// Mitsubishi GX Works2 project: project part 2   PLC: FX3G

// global labels: Global1
VAR_GLOBAL
  switch1 AT X007 : BOOL;
  counter_start_day_result AT CS0 : BOOL;
  creamValue : REAL;  (* ערך למיכל קצפת *)
  creamTank AT D1100 : REAL;  (* ערך למיכל קצפת *)
  chocolateValue : REAL;  (* מיכל שוקולד *)
  chocolateTank AT D1102 : REAL;  (* מיכל השוקולד *)
  biscuitValue : REAL;  (* מיכל ביסקוויטים *)
  biscuitTank AT D1104 : REAL;  (* מיכל ביסקוויטים *)
  zilufTank AT D1112 : REAL;  (* ערך למיכל זילוף *)
END_VAR
VAR_GLOBAL CONSTANT
  zilufValue : REAL;  (* ערך למיכל זילוף *)
  dippingValue : REAL;  (* ערך למיכל טבילה *)
END_VAR
VAR_GLOBAL
  dippingTank AT D1114 : REAL;  (* ערך למיכל טבילה *)
END_VAR
VAR_GLOBAL CONSTANT
  unitsAmount : REAL;  (* כמות קרמבו מוכנים *)
END_VAR
VAR_GLOBAL
  amountDone AT D1118 : REAL;  (* כמות קרמבו מוכנים *)
  switch3 AT X011 : BOOL;  (* העברת הקצפת למיכל זילוף *)
END_VAR
VAR_GLOBAL CONSTANT
  creamInv : REAL := 700;  (* מלאי קצפת *)
END_VAR
VAR_GLOBAL
  courrentCream AT D1106 : REAL;
  curentCream AT D1106 : REAL;
  curentChoclate AT D1108 : REAL;
  curentBiscu AT D1110 : REAL;
END_VAR
VAR_GLOBAL CONSTANT
  chocolateInv : REAL := 500.0;  (* מלאי שוקולד *)
  constBisc : REAL := 6;
  contCream : REAL := 300;
END_VAR
VAR_GLOBAL
  switch4 AT X010 : BOOL;
  switch6 AT X005 : BOOL;
  ReadyToZiluf AT M0 : BOOL;
  TempBelow15 AT M1 : BOOL;
  ingReady AT Y000 : BOOL;
  sen_surface AT X003 : BOOL;
  switch7 AT X001 : BOOL;
  switch8 AT X002 : BOOL;
  under15 AT X001 : BOOL;
  under30 AT X002 : BOOL;
  zilufLight AT Y004 : BOOL;
  sen_camera AT X004 : BOOL;
  checkInv AT X011 : BOOL;  (* האם יש מספיק קצפת וביסקוויטים עבור זילוף *)
  enoughCream AT M111 : BOOL;
  notEnoughCream AT M150 : BOOL;
  enoughBisc AT M112 : BOOL;
  notEnoughBisc AT M151 : BOOL;
  dayStarted AT Y007 : BOOL;
  startDaySwitch AT X007 : BOOL;
  updateInventory AT CS0 : BOOL;
  enoughIng AT M113 : BOOL;
  startFlickering AT M0 : BOOL;
  Timer3 AT TC2 : BOOL;
  Timer1 AT TC1 : BOOL;
END_VAR
VAR_GLOBAL CONSTANT
  fourSeconds : INT := 5;
END_VAR
VAR_GLOBAL
  Timer2 AT TS1 : BOOL;
  Timer4 AT TS2 : BOOL;
  switch10 AT Y000 : BOOL;
  switch11 AT Y001 : BOOL;
  goToMachineB AT M130 : BOOL;
  Timer0 AT TC0 : BOOL;
END_VAR
VAR_GLOBAL CONSTANT
  countFour : INT := 40;
  countHalfSec : INT := 5;
END_VAR
VAR_GLOBAL
  Timer0_0 AT TS0 : BOOL;
  finishedZiluf AT M114 : BOOL;
  finished_fourSec_timer AT TS0 : BOOL;
  startZilufMachine AT X011 : BOOL;
  enoughIng_StartDay AT M115 : BOOL;
  Try_startDay AT M7 : BOOL;
  sample_analogIinput1 AT X006 : BOOL;
  sample AT X006 : BOOL;
END_VAR
VAR_GLOBAL CONSTANT
  normalize_val : INT := 390;
END_VAR
VAR_GLOBAL
  save_analog_val AT D8000 : INT;
  analog_input_chocolate AT D8280 : INT;
  coating AT M116 : BOOL;
  choose_coating_indicator AT M116 : BOOL;
END_VAR
VAR_GLOBAL CONSTANT
  bottom_limit_reg_coat : INT;  (* בדיקה האם הערך גדול מ0 *)
  upper_limit_reg_coat : INT := 5;
END_VAR
VAR_GLOBAL
  biggerThen_0 AT M118 : BOOL;
  smallerThen_5 AT M119 : BOOL;
END_VAR
VAR_GLOBAL CONSTANT
  bottom_limit_double_coat : INT := 6;  (* בדיקה האם הערך גדול 6 *)
END_VAR
VAR_GLOBAL
  biggerThen_6 AT M120 : BOOL;
END_VAR
VAR_GLOBAL CONSTANT
  upper_limit_double_coat : INT := 10;
END_VAR
VAR_GLOBAL
  smallerThen_10 AT M121 : BOOL;
  Regular_coat AT M122 : BOOL;
  Double_coat AT M123 : BOOL;
  successTranfer_toZiluf AT M125 : BOOL;
  chocolateInput AT D1117 : INT;
END_VAR
VAR_GLOBAL CONSTANT
  regularQuantity : REAL := 120;
  doubleQuantity : REAL := 240;
END_VAR
VAR_GLOBAL
  finished_transfer_toDipping AT M124 : BOOL;
  dippingIsOn AT Y003 : BOOL;
  TimerForDipping AT TC3 : BOOL;
END_VAR
VAR_GLOBAL CONSTANT
  countForDipping : INT := 50;
END_VAR
VAR_GLOBAL
  finishedDipping_timer AT TS3 : BOOL;
  enoughChocolate AT M126 : BOOL;  (* מספיק שוקולד לציפוי כפול *)
  notEnoughChocolate AT M128 : BOOL;
  stopDay AT M129 : BOOL;
END_VAR
VAR_GLOBAL CONSTANT
  initVakue : INT;
  initValue : REAL;
END_VAR
VAR_GLOBAL
  Timer_stopDay AT TC5 : BOOL;
END_VAR
VAR_GLOBAL CONSTANT
  countThreeSec : INT := 30;
END_VAR
VAR_GLOBAL
  finished_threeSec_timer AT TS5 : BOOL;
  TimerHalfSec AT TC4 : BOOL;
  finishHalfSec AT TS4 : BOOL;  (* סיום ציפוי *)
  countAgain AT M131 : BOOL;
  TimerHalfSec2 AT TC6 : BOOL;
  finishHalfSec2 AT TS6 : BOOL;
  fictiveLight AT M132 : BOOL;
  check2222 AT Y005 : BOOL;
  check1111 AT Y006 : BOOL;
  turnOnMachinA AT M142 : BOOL;
  stopDay_ind AT M140 : BOOL;
  packOne AT X000 : BOOL;  (* אריזת קרמבו בודד *)
  countPack AT CC1 : BOOL;
END_VAR
VAR_GLOBAL CONSTANT
  count_five : INT := 5;
END_VAR
VAR_GLOBAL
  countPack2 AT CC2 : BOOL;
END_VAR
VAR_GLOBAL CONSTANT
  count_six : INT := 6;
END_VAR
VAR_GLOBAL
  finish_pack5 AT CS1 : BOOL;
  almost_finishPack AT Y002 : BOOL;
  finish_pack6 AT CS2 : BOOL;
  countFinished_units AT CC3 : BOOL;
END_VAR
VAR_GLOBAL CONSTANT
  CountOne : INT := 1;
  add_one : REAL := 1;
END_VAR
VAR_GLOBAL
  Reset_C1 AT CC1 : BOOL;
  Reset_C2 AT CC2 : BOOL;
END_VAR
VAR_GLOBAL CONSTANT
  div_ten : REAL := 10;
  MUL_390 : REAL := 390;
END_VAR
VAR_GLOBAL
  finishDip AT M141 : BOOL;
  analog_output_save AT D8001 : REAL;
  savedAmount AT M133 : BOOL;
  amountDone_div AT D1119 : REAL;  (* כמות קרמבו מוכנים *)
  output_analog AT D8282 : INT;
  amountDone_int AT D1121 : INT;
  readyToStartMachineB AT M144 : BOOL;
  finished_dipping AT M145 : BOOL;
END_VAR

// task Task_01 (event TRUE, interval 0, priority 31): POU_01

PROGRAM POU_01
VAR CONSTANT
  biscInv : REAL := 100;  (* מלאי ביסקוויטים *)
END_VAR
VAR
  analog_input1 : INT;
END_VAR
VAR CONSTANT
  normal_chocolate : INT := 390;
END_VAR
(* structured ladder/FBD written out as ST: instructions are called as NAME(EN, inputs, outputs); _pN, _eN, _tN stand for wires *)
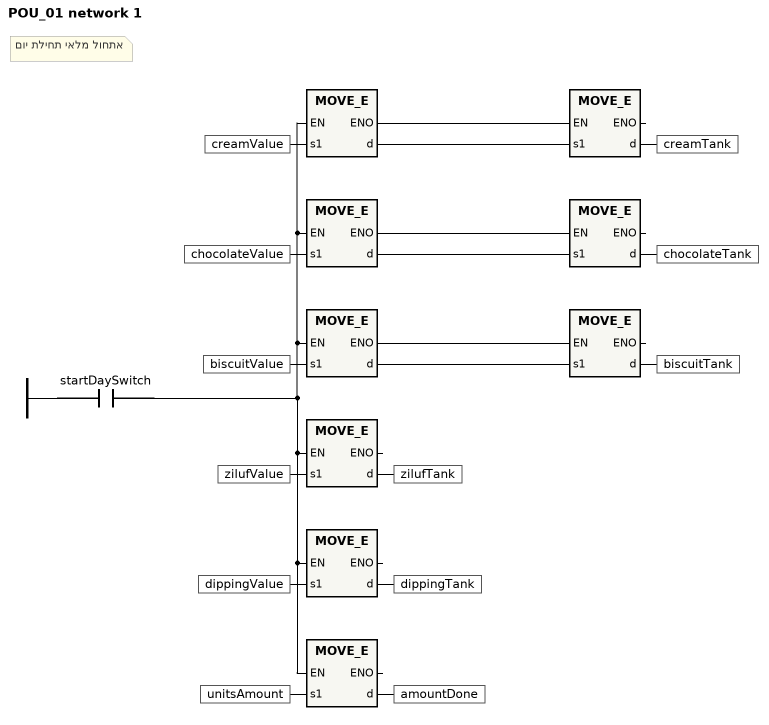
(* network 1 *)
(* אתחול מלאי תחילת יום *)
_e2 := MOVE_E(startDaySwitch, creamValue, _t1);
MOVE_E(_e2, _t1, creamTank);
_e4 := MOVE_E(startDaySwitch, chocolateValue, _t3);
MOVE_E(_e4, _t3, chocolateTank);
_e6 := MOVE_E(startDaySwitch, biscuitValue, _t5);
MOVE_E(_e6, _t5, biscuitTank);
MOVE_E(startDaySwitch, zilufValue, zilufTank);
MOVE_E(startDaySwitch, dippingValue, dippingTank);
MOVE_E(startDaySwitch, unitsAmount, amountDone);
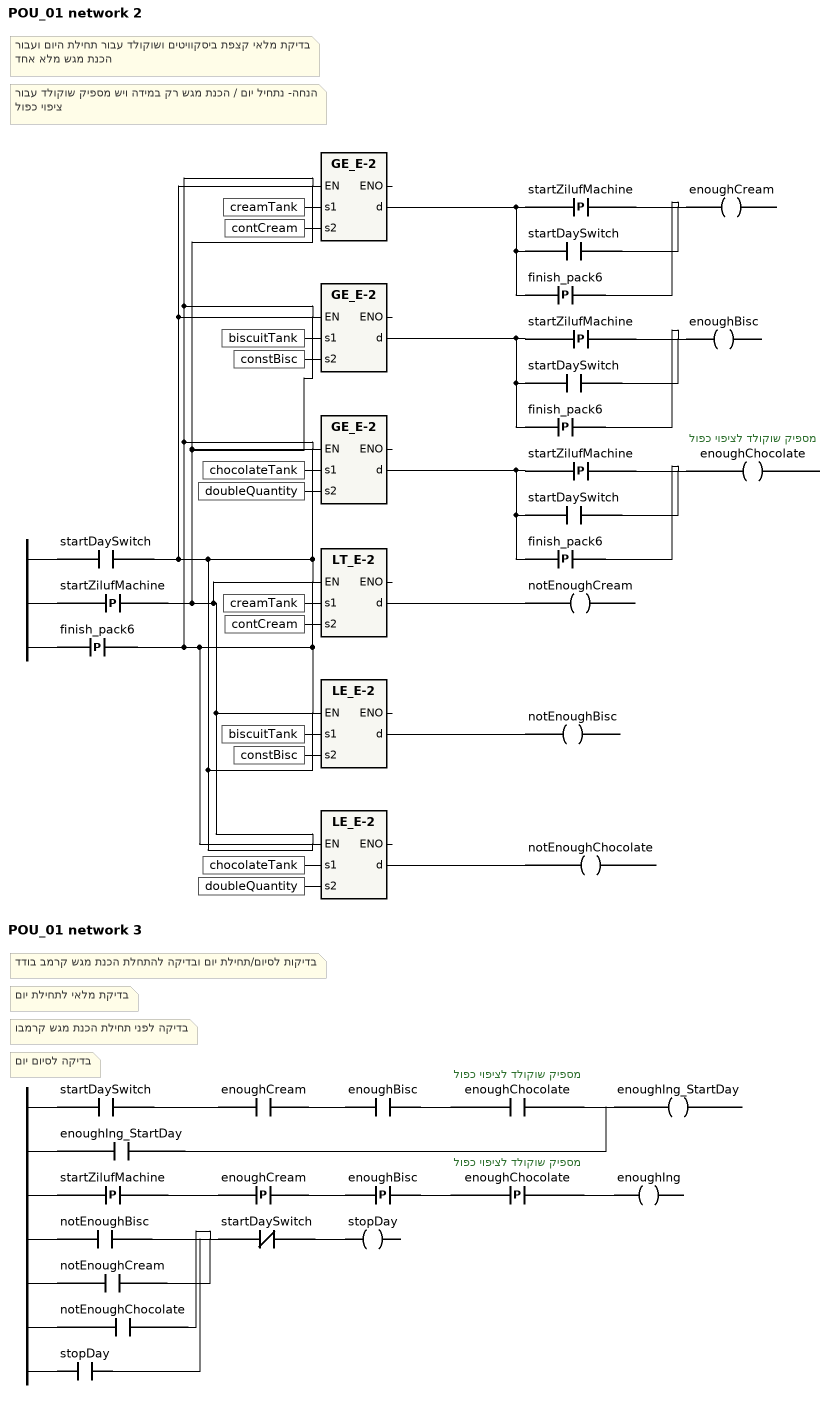
(* network 2 *)
(* בדיקת מלאי קצפת ביסקוויטים ושוקולד עבור תחילת היום ועבור הכנת מגש מלא אחד *)
(* הנחה- נתחיל יום / הכנת מגש רק במידה ויש מספיק שוקולד עבור ציפוי כפול *)
_p1 := startDaySwitch OR LDP(TRUE, startZilufMachine) OR LDP(TRUE, finish_pack6);
GE_E(_p1, creamTank, contCream, _t2);
enoughCream := (_t2 AND LDP(TRUE, startZilufMachine)) OR (_t2 AND startDaySwitch) OR (_t2 AND LDP(TRUE, finish_pack6));
LT_E(_p1, creamTank, contCream, _t3);
notEnoughCream := _t3;
GE_E(_p1, biscuitTank, constBisc, _t4);
enoughBisc := (_t4 AND LDP(TRUE, startZilufMachine)) OR (_t4 AND startDaySwitch) OR (_t4 AND LDP(TRUE, finish_pack6));
LE_E(_p1, biscuitTank, constBisc, _t5);
notEnoughBisc := _t5;
LE_E(_p1, chocolateTank, doubleQuantity, _t6);
notEnoughChocolate := _t6;
GE_E(_p1, chocolateTank, doubleQuantity, _t7);
enoughChocolate := (_t7 AND LDP(TRUE, startZilufMachine)) OR (_t7 AND startDaySwitch) OR (_t7 AND LDP(TRUE, finish_pack6));
(* network 3 *)
(* בדיקות לסיום/תחילת יום ובדיקה להתחלת הכנת מגש קרמב בודד *)
(* בדיקת מלאי לתחילת יום *)
(* בדיקה לפני תחילת הכנת מגש קרמבו *)
(* בדיקה לסיום יום *)
enoughIng_StartDay := (startDaySwitch AND enoughCream AND enoughBisc AND enoughChocolate) OR enoughIng_StartDay;
enoughIng := LDP(TRUE, startZilufMachine) AND LDP(TRUE, enoughCream) AND LDP(TRUE, enoughBisc) AND LDP(TRUE, enoughChocolate);
stopDay := (notEnoughBisc OR notEnoughCream OR notEnoughChocolate OR stopDay) AND NOT startDaySwitch;
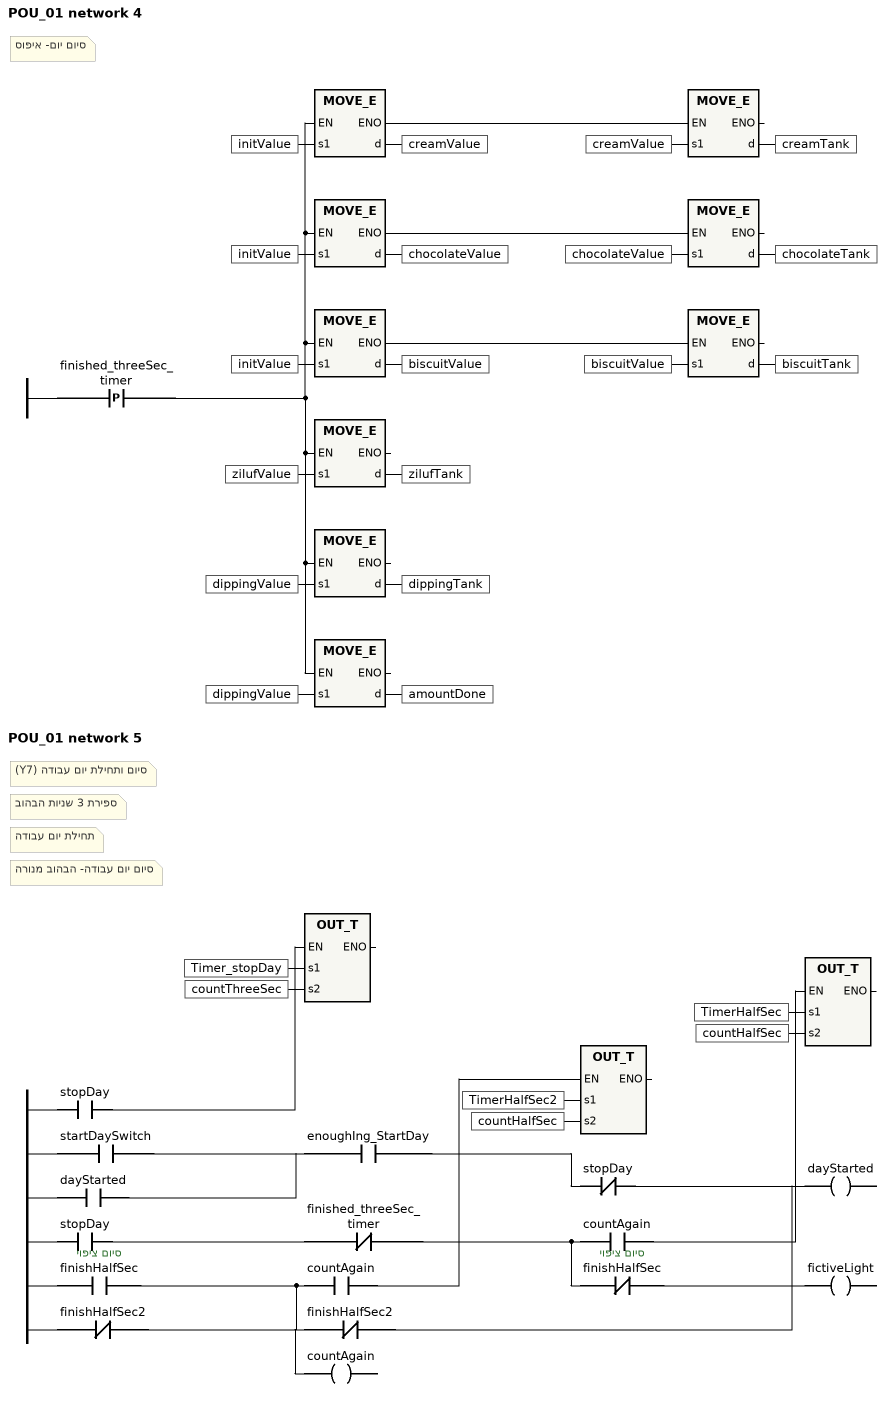
(* network 4 *)
(* סיום יום- איפוס *)
_p1 := LDP(TRUE, finished_threeSec_timer);
_e2 := MOVE_E(_p1, initValue, creamValue);
MOVE_E(_e2, creamValue, creamTank);
_e3 := MOVE_E(_p1, initValue, chocolateValue);
MOVE_E(_e3, chocolateValue, chocolateTank);
_e4 := MOVE_E(_p1, initValue, biscuitValue);
MOVE_E(_e4, biscuitValue, biscuitTank);
MOVE_E(_p1, zilufValue, zilufTank);
MOVE_E(_p1, dippingValue, dippingTank);
MOVE_E(_p1, dippingValue, amountDone);
(* network 5 *)
(* סיום ותחילת יום עבודה (Y7) *)
(* ספירת 3 שניות הבהוב *)
(* תחילת יום עבודה *)
(* סיום יום עבודה- הבהוב מנורה *)
OUT_T(stopDay, Timer_stopDay, countThreeSec);
dayStarted := (((startDaySwitch OR dayStarted) AND enoughIng_StartDay) AND NOT stopDay) OR (finishHalfSec AND NOT finishHalfSec2);
_p1 := stopDay AND NOT finished_threeSec_timer;
OUT_T(_p1 AND countAgain, TimerHalfSec, countHalfSec);
fictiveLight := _p1 AND NOT finishHalfSec;
OUT_T(finishHalfSec AND countAgain, TimerHalfSec2, countHalfSec);
countAgain := NOT finishHalfSec2;
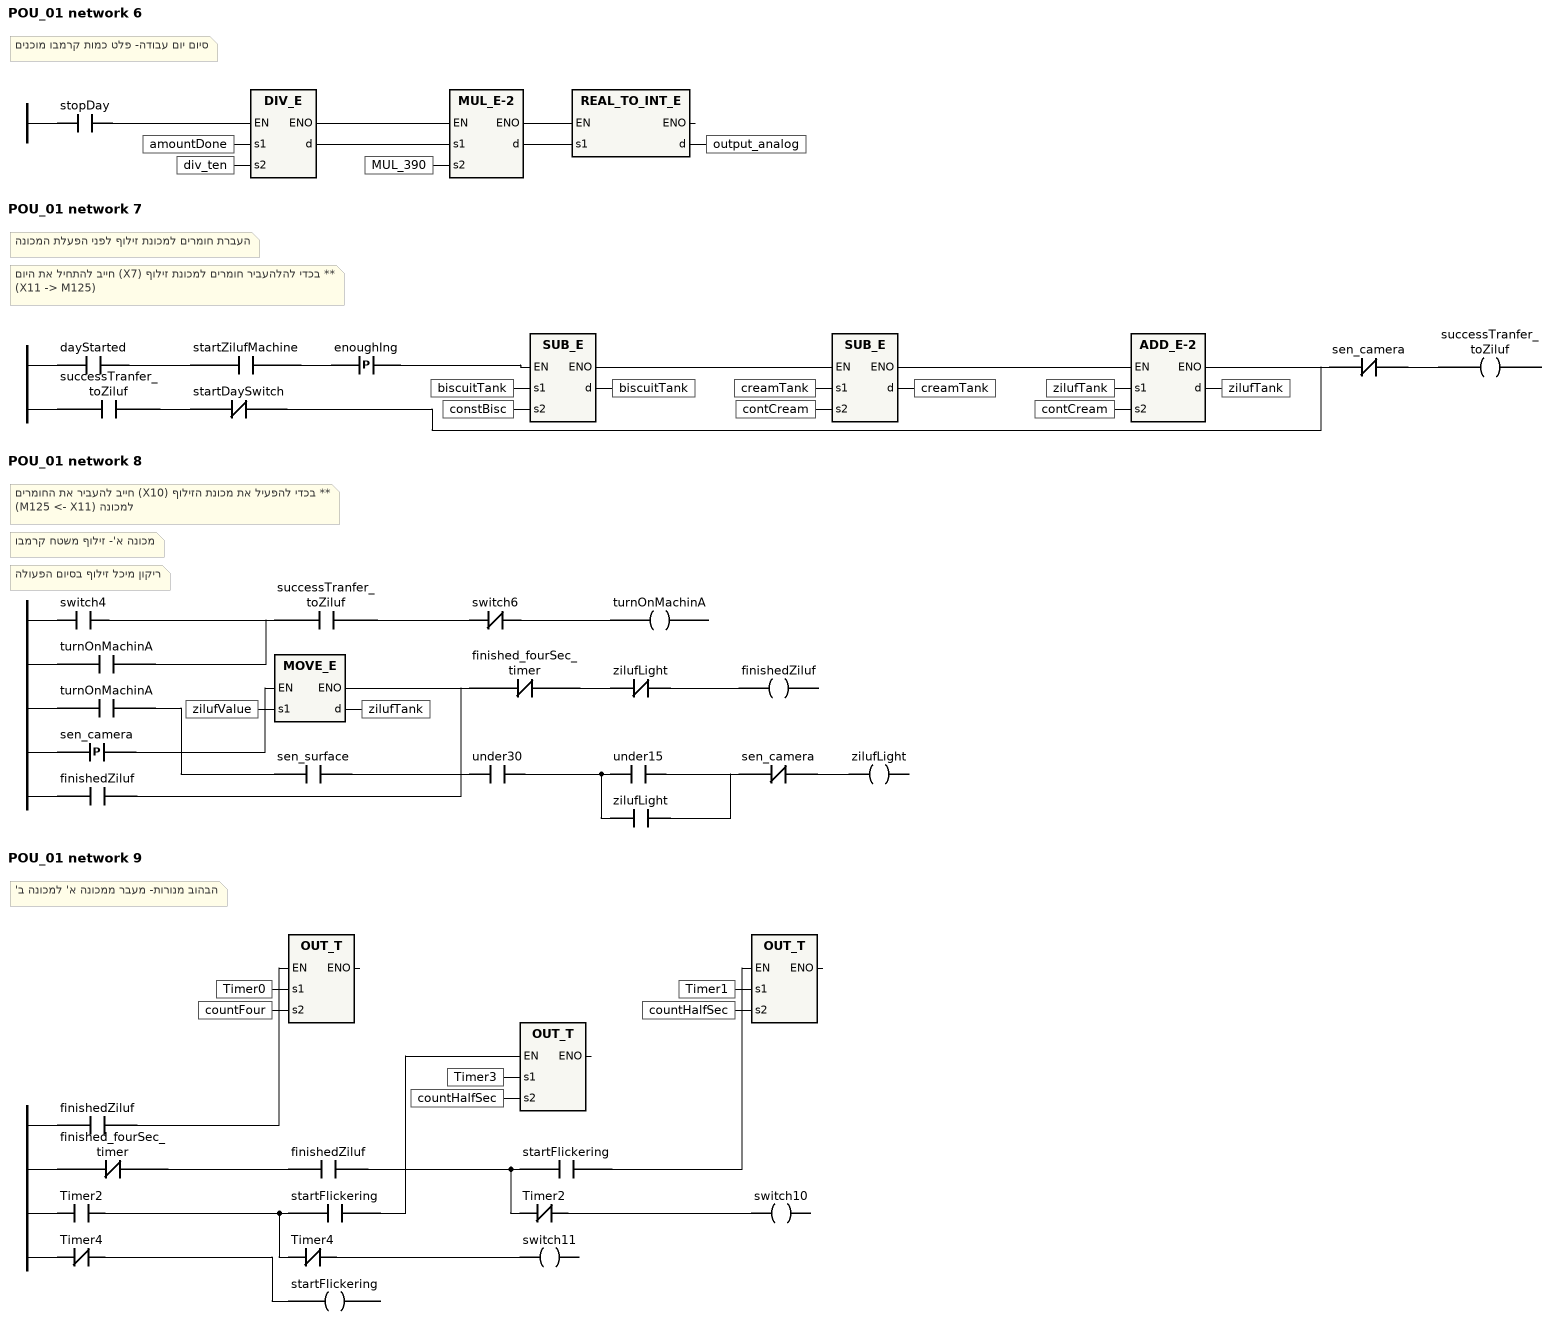
(* network 6 *)
(* סיום יום עבודה- פלט כמות קרמבו מוכנים *)
_e2 := DIV_E(stopDay, amountDone, div_ten, _t1);
_e4 := MUL_E(_e2, _t1, MUL_390, _t3);
REAL_TO_INT_E(_e4, _t3, output_analog);
(* network 7 *)
(* העברת חומרים למכונת זילוף לפני הפעלת המכונה *)
(* ** בכדי להלהעביר חומרים למכונת זילוף (X7) חייב להתחיל את היום  (X11 -> M125) *)
_e1 := SUB_E(dayStarted AND startZilufMachine AND LDP(TRUE, enoughIng), biscuitTank, constBisc, biscuitTank);
_e2 := SUB_E(_e1, creamTank, contCream, creamTank);
_e3 := ADD_E(_e2, zilufTank, contCream, zilufTank);
successTranfer_toZiluf := (_e3 OR (successTranfer_toZiluf AND NOT startDaySwitch)) AND NOT sen_camera;
(* network 8 *)
(* ** בכדי להפעיל את מכונת הזילוף (X10) חייב להעביר את החומרים למכונה (X11 -> M125) *)
(* מכונה א'- זילוף משטח קרמבו *)
(* ריקון מיכל זילוף בסיום הפעולה *)
turnOnMachinA := ((switch4 OR turnOnMachinA) AND successTranfer_toZiluf) AND NOT switch6;
_p1 := turnOnMachinA AND sen_surface AND under30;
zilufLight := ((_p1 AND under15) OR (_p1 AND zilufLight)) AND NOT sen_camera;
_e2 := MOVE_E(LDP(TRUE, sen_camera), zilufValue, zilufTank);
finishedZiluf := ((_e2 OR finishedZiluf) AND NOT finished_fourSec_timer) AND NOT zilufLight;
(* network 9 *)
(* הבהוב מנורות- מעבר ממכונה א' למכונה ב' *)
OUT_T(finishedZiluf, Timer0, countFour);
_p1 := NOT finished_fourSec_timer AND finishedZiluf;
OUT_T(_p1 AND startFlickering, Timer1, countHalfSec);
switch10 := _p1 AND NOT Timer2;
OUT_T(Timer2 AND startFlickering, Timer3, countHalfSec);
switch11 := Timer2 AND NOT Timer4;
startFlickering := NOT Timer4;
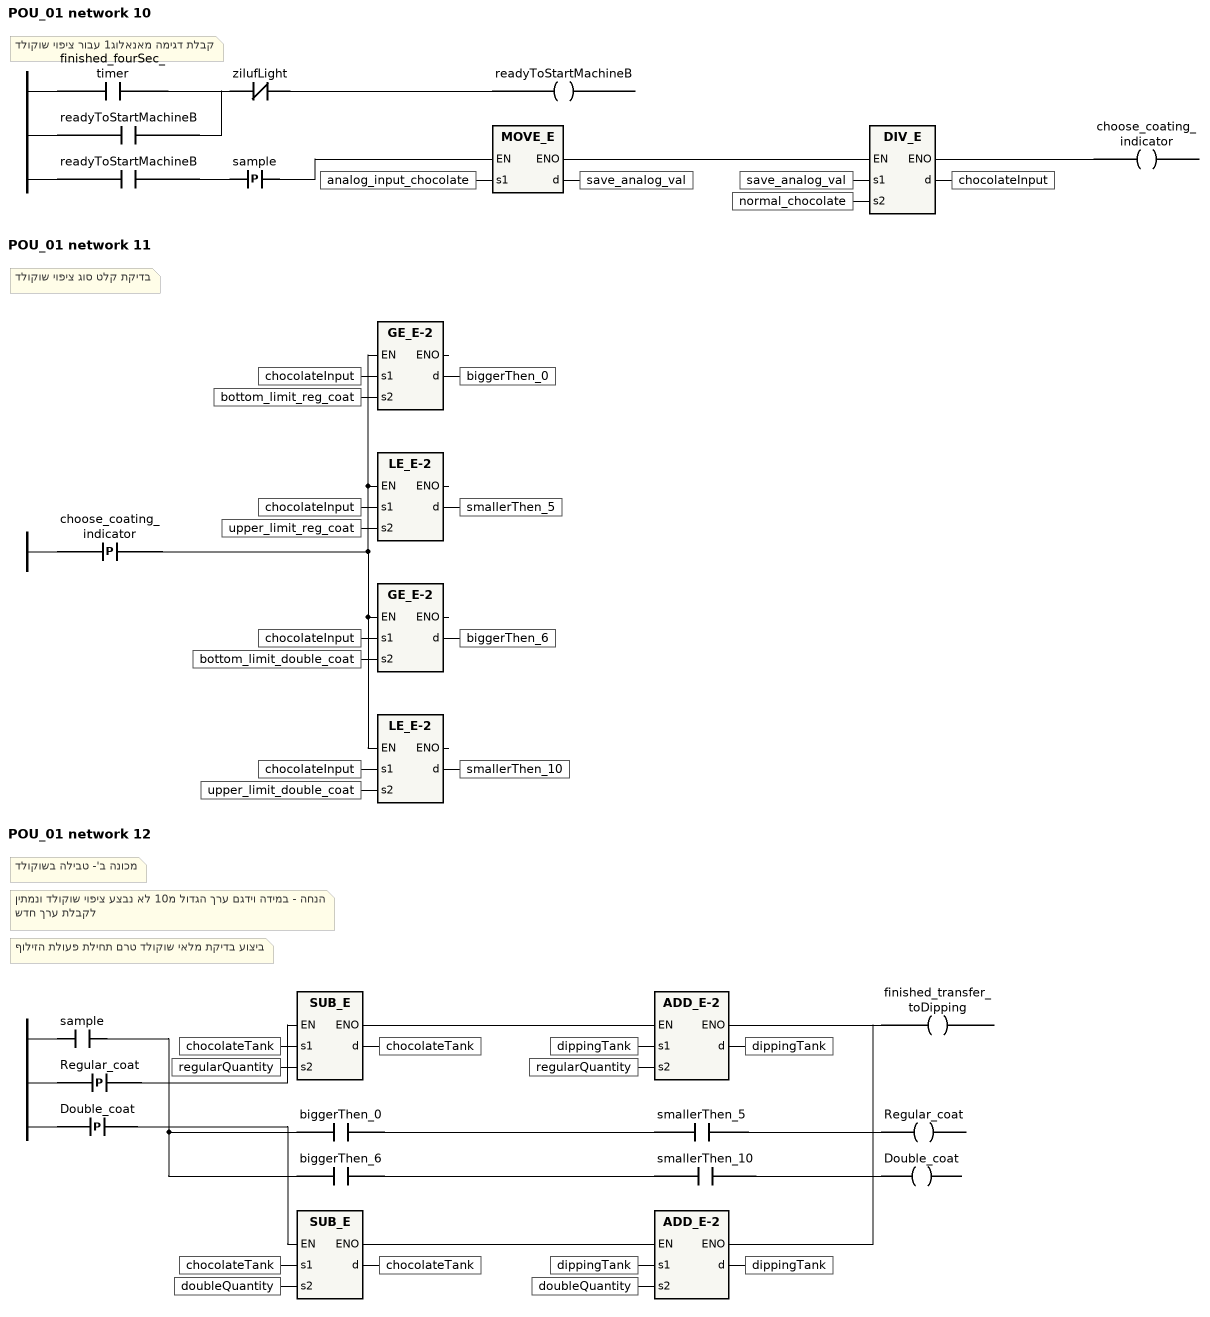
(* network 10 *)
(* קבלת דגימה מאנאלוג1 עבור ציפוי שוקולד *)
readyToStartMachineB := (finished_fourSec_timer OR readyToStartMachineB) AND NOT zilufLight;
_e1 := MOVE_E(readyToStartMachineB AND LDP(TRUE, sample), analog_input_chocolate, save_analog_val);
_e2 := DIV_E(_e1, save_analog_val, normal_chocolate, chocolateInput);
choose_coating_indicator := _e2;
(* network 11 *)
(* בדיקת קלט סוג ציפוי שוקולד *)
_p1 := LDP(TRUE, choose_coating_indicator);
GE_E(_p1, chocolateInput, bottom_limit_reg_coat, biggerThen_0);
LE_E(_p1, chocolateInput, upper_limit_reg_coat, smallerThen_5);
GE_E(_p1, chocolateInput, bottom_limit_double_coat, biggerThen_6);
LE_E(_p1, chocolateInput, upper_limit_double_coat, smallerThen_10);
(* network 12 *)
(* מכונה ב'- טבילה בשוקולד *)
(* הנחה - במידה וידגם ערך הגדול מ10 לא נבצע ציפוי שוקולד ונמתין לקבלת ערך חדש *)
(* ביצוע בדיקת מלאי שוקולד טרם תחילת פעולת הזילוף *)
Regular_coat := sample AND biggerThen_0 AND smallerThen_5;
Double_coat := sample AND biggerThen_6 AND smallerThen_10;
_e1 := SUB_E(LDP(TRUE, Regular_coat), chocolateTank, regularQuantity, chocolateTank);
_e2 := ADD_E(_e1, dippingTank, regularQuantity, dippingTank);
_e3 := SUB_E(LDP(TRUE, Double_coat), chocolateTank, doubleQuantity, chocolateTank);
_e4 := ADD_E(_e3, dippingTank, doubleQuantity, dippingTank);
finished_transfer_toDipping := _e2 OR _e4;
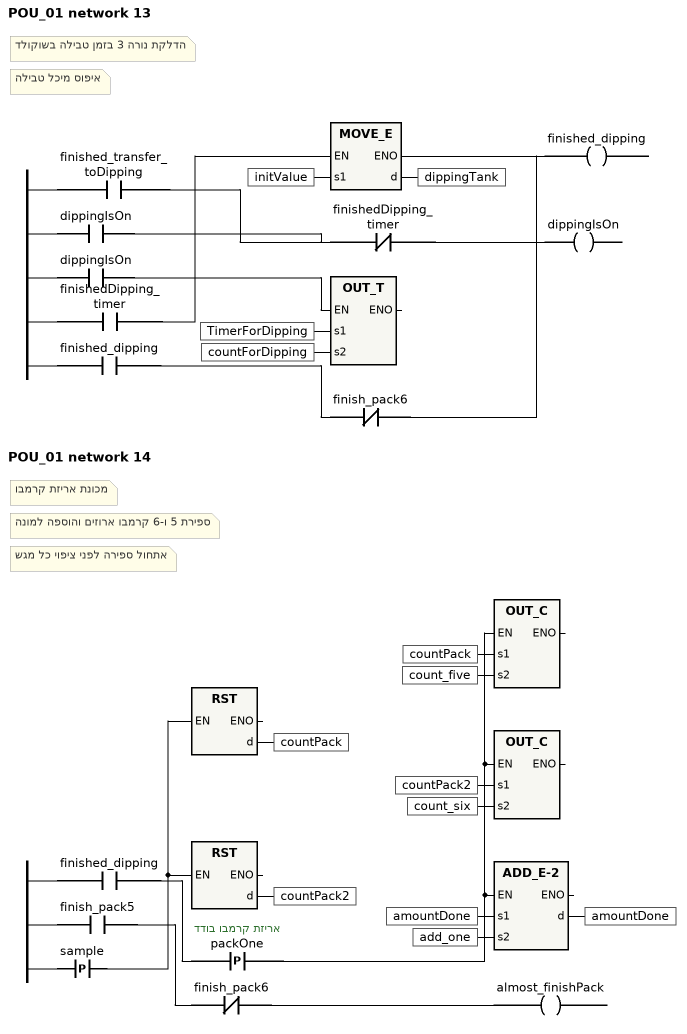
(* network 13 *)
(* הדלקת נורה 3 בזמן טבילה בשוקולד *)
(* איפוס מיכל טבילה *)
dippingIsOn := (finished_transfer_toDipping OR dippingIsOn) AND NOT finishedDipping_timer;
OUT_T(dippingIsOn, TimerForDipping, countForDipping);
_e1 := MOVE_E(finishedDipping_timer, initValue, dippingTank);
finished_dipping := _e1 OR (finished_dipping AND NOT finish_pack6);
(* network 14 *)
(* מכונת אריזת קרמבו *)
(* ספירת 5 ו-6 קרמבו ארוזים והוספה למונה *)
(* אתחול ספירה לפני ציפוי כל מגש *)
_p1 := finished_dipping AND LDP(TRUE, packOne);
OUT_C(_p1, countPack, count_five);
OUT_C(_p1, countPack2, count_six);
ADD_E(_p1, amountDone, add_one, amountDone);
almost_finishPack := finish_pack5 AND NOT finish_pack6;
_p2 := LDP(TRUE, sample);
RST(_p2, countPack);
RST(_p2, countPack2);
END_PROGRAM
